FUNCTION ClearPID 
VAR_INPUT
	enable: BOOL;
	
END_VAR
VAR_IN_OUT
	e0, e1, e2: REAL;
	u0, u1: REAL;
	mea: REAL;
END_VAR
VAR
END_VAR

IF (enable = TRUE) THEN
	e0 := 0;
	e1 := 0;
	e2 := 0;
	u0 := 0;
	u1 := 0;
	mea := 0;
END_IF

END_FUNCTION

(* stored: Version 1.1.0.1, ProductVersion 3.1.4024.3
   POU ClearPID: Id {063cb411-9ab2-4894-b7e6-69372d470e52}, SpecialFunc None *)
